FUNCTION_BLOCK CylinderHSensValve (* Composite Function Block Type *)
  (* Standard: 61499-2 *)
  (* Version 0.0, 5/28/2016, Andrei, nxtControl GmbH, template *)
  PACKAGE Main;
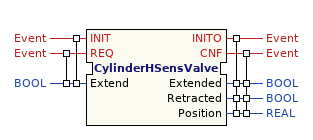
  EVENT_INPUT
    INIT WITH Extend;
    REQ WITH Extend; (* Normal Execution Request *)
  END_EVENT
  EVENT_OUTPUT
    INITO WITH Extended, Retracted, Position;
    CNF WITH Extended, Retracted, Position; (* Execution Confirmation *)
  END_EVENT
  VAR_INPUT
    Extend : BOOL; (* Input event qualifier *)
  END_VAR
  VAR_OUTPUT
    Extended : BOOL; (* Output event qualifier *)
    Retracted : BOOL;
    Position : REAL;
  END_VAR
  FBS
    FB2 : ValveControlSR;
    FB1 : CylinderHSens;
    IThis : CylinderHSensValve_HMI(QI := TRUE);
  END_FBS
  EVENT_CONNECTIONS
    FB2.CNF TO FB1.REQ;
    FB1.CHG TO CNF;
    FB1.INITO TO INITO;
    FB2.INITO TO FB1.INIT;
    INIT TO IThis.INIT;
    REQ TO IThis.REQ;
    IThis.INITO TO FB2.INIT;
    IThis.CNF TO FB2.REQ;
  END_CONNECTIONS
  DATA_CONNECTIONS
    FB2.PV1 TO FB1.PV1;
    FB2.PV2 TO FB1.PV2;
    FB1.Position TO Position;
    FB1.StartSW TO Retracted;
    FB1.EndSW TO Extended;
    IThis.FWD_OUT TO FB2.FWD;
  END_CONNECTIONS
END_FUNCTION_BLOCK
